// TIA Portal V17 export
// export: Created 2023-12-22T15:03:01.5436112Z, ExportSetting WithDefaults, DisplayName Totally Integrated Automation Portal, DisplayVersion V17, DisplayName TIA Portal Openness, DisplayVersion V17, DisplayName TIA Portal Version Control Interface, DisplayVersion V17, DisplayName STEP 7 Professional, DisplayVersion V17, DisplayName STEP 7 Safety, DisplayVersion V17, DisplayName WinCC Advanced, DisplayVersion V17
FUNCTION_BLOCK "AIx"   // FB220, LAD
{ S7_Optimized_Access := 'FALSE' }
VERSION : 0.1
// Signal - PIW код сигнала от датчика
// pulse - частота алгоритма фильтрации
// Result - результат обработки сигнала, формат Real
// stored: AutoNumber false, IsIECCheckEnabled false, SetENOAutomatically false, UDAEnableTagReadback false
   VAR DB_SPECIFIC
      Time_DTL { S7_SetPoint := 'True'} : DTL;
   END_VAR
   VAR_TEMP   // added for the SCL form of the ladder/FBD networks
      _w1 : Bool;
   END_VAR
BEGIN

REGION Network 1: Датчик уровня
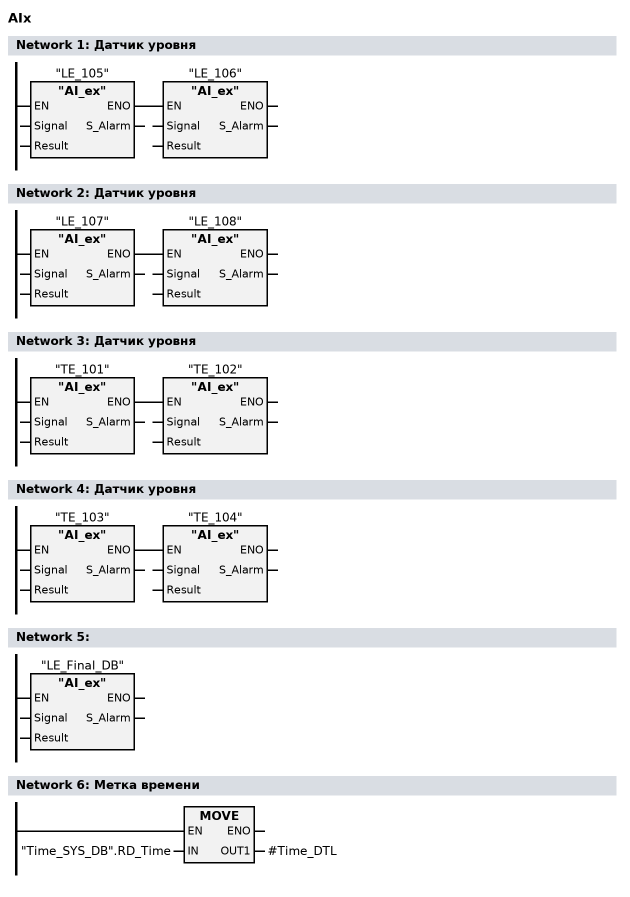
   RUNG wire#powerrail
      "LE_105"(Signal :=, Result :=, S_Alarm =>)
      "LE_106"(Signal :=, Result :=, S_Alarm =>)
   END_RUNG
   // the same network as SCL:
   "LE_105"(ENO => #_w1);   // "AI_ex"
   IF #_w1 THEN
       "LE_106"();   // "AI_ex"
   END_IF;
END_REGION

REGION Network 2: Датчик уровня
   RUNG wire#powerrail
      "LE_107"(Signal :=, Result :=, S_Alarm =>)
      "LE_108"(Signal :=, Result :=, S_Alarm =>)
   END_RUNG
   // the same network as SCL:
   "LE_107"(ENO => #_w1);   // "AI_ex"
   IF #_w1 THEN
       "LE_108"();   // "AI_ex"
   END_IF;
END_REGION

REGION Network 3: Датчик уровня
   RUNG wire#powerrail
      "TE_101"(Signal :=, Result :=, S_Alarm =>)
      "TE_102"(Signal :=, Result :=, S_Alarm =>)
   END_RUNG
   // the same network as SCL:
   "TE_101"(ENO => #_w1);   // "AI_ex"
   IF #_w1 THEN
       "TE_102"();   // "AI_ex"
   END_IF;
END_REGION

REGION Network 4: Датчик уровня
   RUNG wire#powerrail
      "TE_103"(Signal :=, Result :=, S_Alarm =>)
      "TE_104"(Signal :=, Result :=, S_Alarm =>)
   END_RUNG
   // the same network as SCL:
   "TE_103"(ENO => #_w1);   // "AI_ex"
   IF #_w1 THEN
       "TE_104"();   // "AI_ex"
   END_IF;
END_REGION

REGION Network 5
   RUNG wire#powerrail
      "LE_Final_DB"(Signal :=, Result :=, S_Alarm =>)
   END_RUNG
   // the same network as SCL:
   "LE_Final_DB"();   // "AI_ex"
END_REGION

REGION Network 6: Метка времени
   RUNG wire#powerrail
      Move(in := "Time_SYS_DB".RD_Time, out1 => #Time_DTL)
   END_RUNG
   // the same network as SCL:
   #Time_DTL := "Time_SYS_DB".RD_Time;
END_REGION
END_FUNCTION_BLOCK
